TYPE ST_DigitalLamp :
STRUCT
	PushButton: BOOL;	
	ToggleButton: BOOL;
	Status: BOOL;

END_STRUCT
END_TYPE

(* stored: Version 1.1.0.1, ProductVersion 3.1.4024.13
   DUT ST_DigitalLamp: Id {533ecbba-df96-4d7b-b11b-308b850fcea2} *)
